{attribute 'qualified_only'}
{attribute 'strict'}
TYPE ABBLINKIN_AUTH_HEADER_VALUE :
(
	NONE,
	BASIC,
	DIGEST
);
END_TYPE

(* stored: Version 1.1.0.1, ProductVersion 3.1.4024.12
   DUT ABBLINKIN_AUTH_HEADER_VALUE: Id {99690849-bea9-4839-8bf4-6dc76e95b60f} *)
